// TwinCAT 3 PLC project MAS418_PLC
// ProgramVersion: 3.1.4024.0
// libraries:
//   Tc2_Standard, * (Beckhoff Automation GmbH)
//   Tc2_System, * (Beckhoff Automation GmbH)
//   Tc3_Module, * (Beckhoff Automation GmbH)
//   VisuDialogs, * (System)
//   VisuSymbols,3.5.10.0,System
// project tree:
//   / GlobalTextList.TcGTLO, PlcTask.TcTTO, Visualization Manager.TcVMO (not stored)
//   POUs/ MAIN.TcPOU
//   VISUs/ HMI.TcVIS
// real-time tasks:
//   TASK PlcTask: cycle T#10ms, priority 20, ADS port 350

CONFIGURATION MAS418_PLC
    RESOURCE PLC ON TwinCAT3
        TASK PlcTask(INTERVAL := T#10ms, PRIORITY := 20);
        PROGRAM MAIN WITH PlcTask : MAIN;
    END_RESOURCE
END_CONFIGURATION

// ---- POUs/MAIN.TcPOU
PROGRAM MAIN
VAR
	bEnable 		: BOOL;
	bStart  		: BOOL;
	nINT			: INT;
	nUINT			: UINT;
	fREAL			: REAL;
	sPowerStatus	: STRING;
	nFloatConversion : INT;
	fFloatConversion : LREAL;
	nFloatcon2		 : INT;
	fFloatcon2		 : LREAL :=10.1;
END_VAR

bEnable := bStart;

nINT := -32768;
nUINT := 65535;
fREAL := 255.255;

sPowerStatus := 'Power OFF';

fFloatConversion := nFloatConversion;

nFloatcon2 := LREAL_TO_INT(fFloatcon2);

END_PROGRAM

// ---- GlobalTextList.TcGTLO
TEXTLIST GlobalTextList
  928 = 'BOOL'
  697 = 'BOOL %i'
  891 = 'DataTypeTesting'
  954 = 'HMI'
  751 = 'INT'
  454 = 'INT %i'
  4 = 'Power ON'
  74 = 'REAL'
  427 = 'REAL %f'
  471 = 'REAL %i'
  931 = 'STRING'
  124 = 'STRING %s'
  234 = 'UINT'
  169 = 'UINT %i'
END_TEXTLIST

// ---- VISUs/HMI.TcVIS
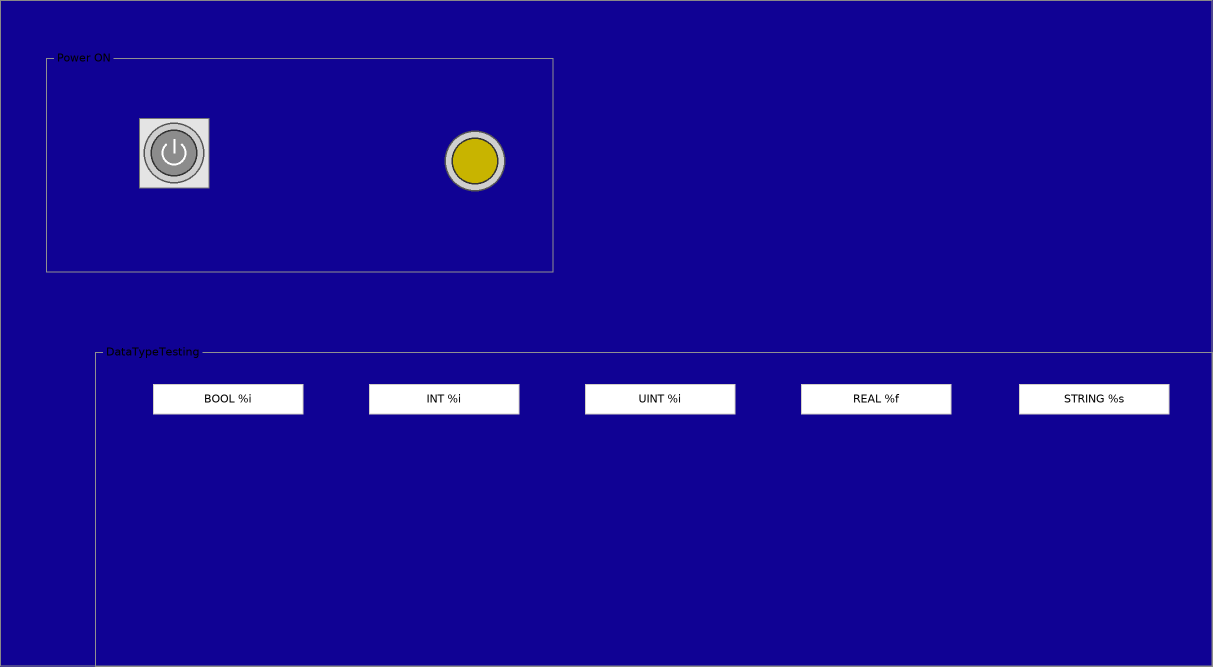
VISUALIZATION HMI  // 1213x667
    GroupBox (46,50 507x222), "Power ON"
        Lamp1 (394,76 70x70), variable: MAIN.bEnable, style: Lamp-Lamp1-Yellow
        PowerSwitch (93,68 70x70), variable: MAIN.bStart, behaviour: TOGGLE, style: Switch-PowerSwitch-Gray
    GroupBox (95,344 1118x323), "DataTypeTesting"
        Textfield (58,40 150x30), "BOOL %i", text variable: MAIN.bEnable
            toggle MAIN.bEnable
        Textfield (274,40 150x30), "INT %i", text variable: MAIN.nINT
        Textfield (924,40 150x30), "STRING %s", text variable: MAIN.sPowerStatus
            OnMouseDown: write the text variable via Default
        Textfield (490,40 150x30), "UINT %i", text variable: MAIN.nUINT
        Textfield (706,40 150x30), "REAL %f", text variable: MAIN.fREAL
            OnMouseDown: write the text variable via Default, min -5000, max 5000
END_VISUALIZATION
